// TIA Portal V18 export
VAR_GLOBAL   // PLC tag table "Default tag table"
   Tag_1 AT %M0.0 : Bool;
   System_Byte AT %MB1 : Byte;
   FirstScan AT %M1.0 : Bool;
   DiagStatusUpdate AT %M1.1 : Bool;
   AlwaysTRUE AT %M1.2 : Bool;
   AlwaysFALSE AT %M1.3 : Bool;
   Clock_Byte AT %MB0 : Byte;
   Clock_10Hz AT %M0.0 : Bool;
   Clock_5Hz AT %M0.1 : Bool;
   "Clock_2.5Hz" AT %M0.2 : Bool;
   Clock_2Hz AT %M0.3 : Bool;
   "Clock_1.25Hz" AT %M0.4 : Bool;
   Clock_1Hz AT %M0.5 : Bool;
   "Clock_0.625Hz" AT %M0.6 : Bool;
   "Clock_0.5Hz" AT %M0.7 : Bool;
   Tag_2 AT %M10.0 : Bool;
   Tag_3 AT %MW20 : Word;
   Tag_4 AT %M20.1 : Bool;
   Tag_5 AT %MD20 : Real;
   Tag_6 AT %M10.7 : Bool;
   Tag_7 AT %MD30 : DWord;
   Tag_8 AT %M10.5 : Bool;
END_VAR
